// TIA Portal V19 export
TYPE "Straightener_Manager"
   STRUCT
      Feed : "PositioningMachine_Manager";
      Lift_Entry : "ValveMachine_Manager";
      Lift_Exit : "ValveMachine_Manager";
   END_STRUCT;
END_TYPE
